Fanuc KAREL source: kt00752.KL

-- PROVISIONAL review KL for V770-1; original PC SHA256 545676e773b6f72d960f2f57452115c14ddbaf901ec4d86e7978729e3b18340d
-- Incomplete behavior may be omitted. Consult companion uncertainty JSON. Do not deploy.
PROGRAM KT00752
%NOLOCKGROUP
VAR
  OUT : INTEGER
-- UNRESOLVED_DECL Y1 type=002018
-- UNRESOLVED_DECL Y2 type=002018
BEGIN
  -- UNRESOLVED_PC offsets 5-19; opcodes 2E,22,9D,33,B2
  -- UNRESOLVED_PC offsets 24-38; opcodes 2E,22,9D,33,B2
  -- UNRESOLVED_PC offsets 43-57; opcodes 2E,22,9D,33,B2
  -- UNRESOLVED_PC offsets 62-76; opcodes 2E,22,9D,33,B2
  -- UNRESOLVED_PC offsets 81-97; opcodes 22,9D,33,B1,50,23
  -- UNRESOLVED_PC offsets 102-106; opcodes 7F
END KT00752
